KUKA KRL program: TestContSpiral.src, TestContSpiral.dat

--- TestContSpiral.src ---
&ACCESS RVEO
&REL 64
DEF TestContSpiral()
   ;FOLD DECL
      DECL ST_Dim3 stHole
      DECL POS xHole,xAboveHole,xAboveTable
      DECL POS xAboveWall,xOffset
      DECL INT iWall,iPoint,iPointSize
   ;ENDFOLD (DECL)

   stHole = {rX 600,rY 400,rZ 100}
   geProfile = #Frame90

   ;FOLD INI
      xHole = xAboveTableIni
      xHole.X = stHole.rX
      xHole.Y = stHole.rY
      xHole.Z = stHole.rZ

      xAboveTable = xAboveTableIni
      xAboveTable.X = stHole.rX
      xAboveHole = xAboveHoleOffset:xHole

      iPointSize = rHoleDepth/rCycleStepZ * iCycleSize
   ;ENDFOLD (INI)

   ChangeStation(#MillVertRight)

   BAS(#INITMOV)
   SetBaseTool(#MillTable,#Cutter8)

   SetVel(#SpindleIdle)
   LIN xAboveTable C_DIS

   SetVel(#SpindleIdle)
   BAS(#ACC_CP,10)
   LIN xAboveHole C_DIS

   FOR iPoint=1 TO iPointSize STEP 1
      xOffset = GetSpiralOffset(iPoint,iPointSize)
      LIN xOffset:xHole C_DIS
   ENDFOR

   SetVel(#SpindleIdle)
   LIN xAboveHole C_DIS
   LIN xAboveTable C_DIS

   ChangeStation(#HomePos)

END

DEFFCT POS GetSpiralOffset(iPoint:IN,iPointSize:IN)
   ;FOLD DECL
      DECL POS xOffset
      DECL REAL rPathRadius,rDepthStep,rAngle
      DECL INT iPoint,iPointSize
   ;ENDFOLD (DECL)

   rAngle = (iPoint-1) * 360.0/iCycleSize
   rDepthStep = rHoleDepth/iPointSize
   rPathRadius = (rHoleDiameter-grFiCutter8)/2

   xOffset = $NULLFRAME
   xOffset.X = rPathRadius * COS(rAngle)
   xOffset.Y = rPathRadius * SIN(rAngle)
   xOffset.Z = iPoint*rDepthStep

   RETURN xOffset

ENDFCT

--- TestContSpiral.dat ---
&ACCESS RVEO
&REL 64
DEFDAT TestContSpiral

   DECL CONST POS xAboveTableIni = {x 0,y 200,z 120,a 0,b 0,c 0}

   DECL CONST REAL rHoleDiameter = 200.0
   DECL CONST REAL rCycleStepZ = 20.0
   DECL CONST INT iCycleSize = 4
   DECL CONST REAL rHoleDepth = 100.0

   DECL CONST POS xAboveHoleOffset = {x 0,y 0,z 50,a 0,b 0,c 0}
   DECL CONST POS xAboveWallOffset = {x 0,y 0,z 5,a 0,b 0,c 0}
   DECL CONST POS xInsideWallOffset = {x 0,y 0,z -4,a 0,b 0,c 0}

ENDDAT
